// TwinCAT 3 PLC project Manual
// ProgramVersion: 3.1.4023.0
// libraries:
//   Tc2_Standard, * (Beckhoff Automation GmbH)
//   Tc2_System, * (Beckhoff Automation GmbH)
//   Tc3_Module, * (Beckhoff Automation GmbH)
// project tree:
//   / Gestor de visualización.TcVMO (not stored), GlobalTextList.TcGTLO (not stored), PlcTask.TcTTO
//   POUs/ FB_Estacion.TcPOU, MAIN.TcPOU (not stored)
//   VISUs/ Visualization.TcVIS
// real-time tasks:
//   TASK PlcTask: cycle T#10ms, priority 20, ADS port 350
// I/O:
//   DEVICE Device 1 (EtherCAT), AmsNetId 5.67.250.180.2.1
//     Term 1 (EK1200) [EK1200-5000 EtherCAT Power supply (2A E-Bus)]
//       Term 2 (EL1008) [EL1008 8Ch. Dig. Input 24V, 3ms]
//       Term 3 (EL1008) [EL1008 8Ch. Dig. Input 24V, 3ms]
//       Term 4 (EL2008) [EL2008 8Ch. Dig. Output 24V, 0.5A]
//       Term 5 (EL2008) [EL2008 8Ch. Dig. Output 24V, 0.5A]
//       Term 6 (EL1008) [EL1008 8Ch. Dig. Input 24V, 3ms]
//       Term 7 (EL1008) [EL1008 8Ch. Dig. Input 24V, 3ms]
//       Term 8 (EL2008) [EL2008 8Ch. Dig. Output 24V, 0.5A]
//       Term 9 (EL2008) [EL2008 8Ch. Dig. Output 24V, 0.5A]
//       Term 10 (EL9011) [EL9011 End Terminal]
//   DEVICE Device 3 (RT-Ethernet Protocol), AmsNetId 5.67.250.180.4.1
//   DEVICE Device 2 (NOV-DP-RAM)
// variable links:
//   FMS_201_Manual/FMS_201_Manual Instance <-> Device 1 (EtherCAT)/Term 1 (EK1200)/Term 2 (EL1008)
//     PlcTask Inputs/MAIN.ESTACION.EstacionConectada <-> Channel 5/EstacionConectada
//     PlcTask Inputs/MAIN.ESTACION.PaleCodigoBit0 <-> Channel 7/PaleCodigoBit0
//     PlcTask Inputs/MAIN.ESTACION.PaleCodigoBit1 <-> Channel 8/PaleCodigoBit1
//     PlcTask Inputs/MAIN.ESTACION.PalePresencia <-> Channel 6/PalePresencia
//     PlcTask Inputs/MAIN.ESTACION.PulsadorEmergencia <-> Channel 1/PulsadorEmergencia
//     PlcTask Inputs/MAIN.ESTACION.PulsadorMarcha <-> Channel 3/PulsadorMarcha
//     PlcTask Inputs/MAIN.ESTACION.PulsadorParada <-> Channel 4/PulsadorParada
//     PlcTask Inputs/MAIN.ESTACION.SelectorManual <-> Channel 2/SelectorManual
//   FMS_201_Manual/FMS_201_Manual Instance <-> Device 1 (EtherCAT)/Term 1 (EK1200)/Term 3 (EL1008)
//     PlcTask Inputs/MAIN.ESTACION.DetectorPresion <-> Channel 2/DetectorPresion
//     PlcTask Inputs/MAIN.ESTACION.PaleCodigoBit2 <-> Channel 1/PaleCodigoBit2
//   FMS_201_Manual/FMS_201_Manual Instance <-> Device 1 (EtherCAT)/Term 1 (EK1200)/Term 4 (EL2008)
//     PlcTask Outputs/MAIN.ESTACION.CintaMotorActiva <-> Channel 5/CintaMotorActiva
//     PlcTask Outputs/MAIN.ESTACION.CintaMotorInvierte <-> Channel 6/CintaMotorInvierte
//     PlcTask Outputs/MAIN.ESTACION.CintaRetenedorBaja <-> Channel 7/CintaRetenedorBaja
//     PlcTask Outputs/MAIN.ESTACION.CintaSeparadorSube <-> Channel 8/CintaSeparadorSube
//     PlcTask Outputs/MAIN.ESTACION.DesconectaEstacion <-> Channel 1/DesconectaEstacion
//     PlcTask Outputs/MAIN.ESTACION.LamparaAlarma <-> Channel 2/LamparaAlarma
//     PlcTask Outputs/MAIN.ESTACION.LamparaFaltaMaterial <-> Channel 4/LamparaFaltaMaterial
//     PlcTask Outputs/MAIN.ESTACION.LamparaMarcha <-> Channel 3/LamparaMarcha
//   FMS_201_Manual/FMS_201_Manual Instance <-> Device 1 (EtherCAT)/Term 1 (EK1200)/Term 5 (EL2008)
//     PlcTask Outputs/MAIN.ESTACION.AvisadorSonoro <-> Channel 1/AvisadorSonoro
//   FMS_201_Manual/FMS_201_Manual Instance <-> Device 1 (EtherCAT)/Term 1 (EK1200)/Term 6 (EL1008)
//     PlcTask Inputs/MAIN.ESTACION.AlimentadorDetras <-> Channel 8/AlimentadorDetras
//     PlcTask Inputs/MAIN.ESTACION.DescargadorDelante <-> Channel 2/DescargadorDelante
//     PlcTask Inputs/MAIN.ESTACION.DescargadorDetras <-> Channel 1/DescargadorDetras
//     PlcTask Inputs/MAIN.ESTACION.DesplazadorDetras <-> Channel 7/DesplazadorDetras
//     PlcTask Inputs/MAIN.ESTACION.VerificadorAbajo <-> Channel 6/VerificadorAbajo
//     PlcTask Inputs/MAIN.ESTACION.VerificadorArriba <-> Channel 5/VerificadorArriba
//     PlcTask Inputs/MAIN.ESTACION.VerticalAbajo <-> Channel 4/VerticalAbajo
//     PlcTask Inputs/MAIN.ESTACION.VerticalArriba <-> Channel 3/VerticalArriba
//   FMS_201_Manual/FMS_201_Manual Instance <-> Device 1 (EtherCAT)/Term 1 (EK1200)/Term 7 (EL1008)
//     PlcTask Inputs/MAIN.ESTACION.AlimentadorDelante <-> Channel 1/AlimentadorDelante
//     PlcTask Inputs/MAIN.ESTACION.PresenciaBaseAlimentador <-> Channel 3/PresenciaBaseAlimentador
//     PlcTask Inputs/MAIN.ESTACION.VacioDescargador <-> Channel 2/VacioDescargador
//   FMS_201_Manual/FMS_201_Manual Instance <-> Device 1 (EtherCAT)/Term 1 (EK1200)/Term 8 (EL2008)
//     PlcTask Outputs/MAIN.ESTACION.AlimentadorAdelante <-> Channel 7/AlimentadorAdelante
//     PlcTask Outputs/MAIN.ESTACION.DescargadorAdelante <-> Channel 1/DescargadorAdelante
//     PlcTask Outputs/MAIN.ESTACION.DescargadorAtras <-> Channel 2/DescargadorAtras
//     PlcTask Outputs/MAIN.ESTACION.DescargadorBaja <-> Channel 3/DescargadorBaja
//     PlcTask Outputs/MAIN.ESTACION.DesplazadorAdelante <-> Channel 6/DesplazadorAdelante
//     PlcTask Outputs/MAIN.ESTACION.EyectorSucciona <-> Channel 8/EyectorSucciona
//     PlcTask Outputs/MAIN.ESTACION.RechazadorAdelante <-> Channel 4/RechazadorAdelante
//     PlcTask Outputs/MAIN.ESTACION.VerificadorBaja <-> Channel 5/VerificadaorBaja

CONFIGURATION Manual
    RESOURCE PLC ON TwinCAT3
        TASK PlcTask(INTERVAL := T#10ms, PRIORITY := 20);
        PROGRAM MAIN WITH PlcTask : MAIN;
    END_RESOURCE
END_CONFIGURATION

// ---- POUs/FB_Estacion.TcPOU
FUNCTION_BLOCK FB_Estacion
VAR_INPUT
END_VAR
VAR_OUTPUT
	//Parametros de salida
	PaleCodigo: BYTE;
END_VAR
VAR
	//Entradas comunes
	PulsadorEmergencia AT %I*: BOOL;
	SelectorManual AT %I*: BOOL;
	PulsadorMarcha AT %I*: BOOL;
	PulsadorParada AT %I*: BOOL := TRUE; //Contacto normalmente cerrado
	EstacionConectada AT %I*: BOOL := TRUE;
	DetectorPresion AT %I*: BOOL := TRUE;
	
	PalePresencia AT %I*: BOOL;
	PaleCodigoBit0 AT %I*: BOOL;
	PaleCodigoBit1 AT %I*: BOOL;
	PaleCodigoBit2 AT %I*: BOOL;
	
	//Entradas específicas
	//Cilindros
	DescargadorDetras AT %I*: BOOL;
	DescargadorDelante AT %I*: BOOL;
	VerticalArriba AT %I*: BOOL;
	VerticalAbajo AT %I*: BOOL;
	VerificadorArriba AT %I*: BOOL;
	VerificadorAbajo AT %I*: BOOL;
	DesplazadorDetras AT %I*: BOOL;
	AlimentadorDetras AT %I*: BOOL;
	AlimentadorDelante AT %I*: BOOL;
	
	VacioDescargador AT %I*: BOOL;
	PresenciaBaseAlimentador AT %I*: BOOL;
	
	//Salidas comunes
	DesconectaEstacion AT %Q*: BOOL;
	LamparaAlarma AT %Q*: BOOL;
	LamparaMarcha AT %Q*: BOOL;
	AvisadorSonoro AT %Q*: BOOL;
	
	CintaMotorActiva AT %Q*: BOOL;
	CintaMotorInvierte AT %Q*: BOOL;
	CintaRetenedorBaja AT %Q*: BOOL;
	CintaSeparadorSube AT %Q*: BOOL;
	
	//Salidas específicas
	DescargadorAtras AT %Q*: BOOL;
	DescargadorAdelante AT %Q*: BOOL;
	DescargadorBaja AT %Q*: BOOL;
	RechazadorAdelante AT %Q*: BOOL;
	VerificadorBaja AT %Q*: BOOL;
	DesplazadorAdelante AT %Q*: BOOL;
	AlimentadorAdelante AT %Q*: BOOL;
	EyectorSucciona AT %Q*: BOOL;
	
	
	
END_VAR

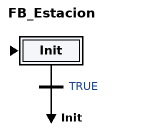
INITIAL_STEP Init:
END_STEP
TRANSITION FROM Init TO Init
    := TRUE;
END_TRANSITION

END_FUNCTION_BLOCK

// ---- VISUs/Visualization.TcVIS
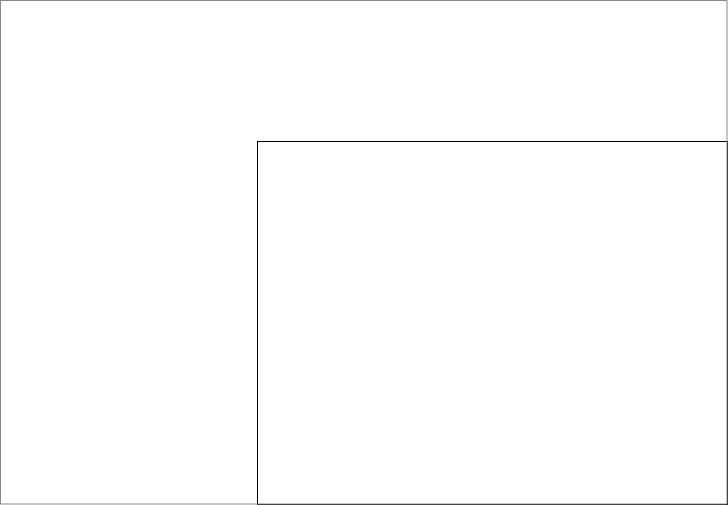
VISUALIZATION Visualization  // 728x505
    Rectangle (257,141 471x364)
END_VISUALIZATION
